(* IEC 61131-3 sources: Industry-PLC-LLM/data/PLCBEAD_repo/PLCBEAD_PLCEmbed-main/PLC-BEAD/Source/GEB/DEAD_ZONE2, 1 file *)

(* ---- DEAD_ZONE2.ST ---- *)
FUNCTION_BLOCK DEAD_ZONE2
	VAR_INPUT
		X :	REAL;
		L :	REAL;
	END_VAR

	VAR_OUTPUT
		Y :	REAL;
	END_VAR

	IF ABS(X) > L THEN
		Y := X;
	ELSIF Y > 0.0 THEN
		Y := L;
	ELSE
		Y := -L;
	END_IF;
END_FUNCTION_BLOCK

PROGRAM program0
  VAR
    LocalVar0 : REAL;
	LocalVaR1  : REAL;
	LocalOUT  : REAL;
	func_block : DEAD_ZONE2;
  END_VAR
	func_block.X  := LocalVar0;
	func_block.L  := LocalVaR1 ;
	func_block();
	LocalOUT := func_block.Y;
END_PROGRAM
